(* PLC project SafeLOGIC-1, BrAutomation SafeDESIGNER  4.2.2.18 *)
(* stored: companyURL http://www.br-automation.com, creationDateTime Wed Apr 19 11:53:29 2017 *)

PROGRAM Main
  VAR  (* added by the conversion: wires and edge detectors of the diagram *)
    _AND_S80_OUT : ANY;
  END_VAR

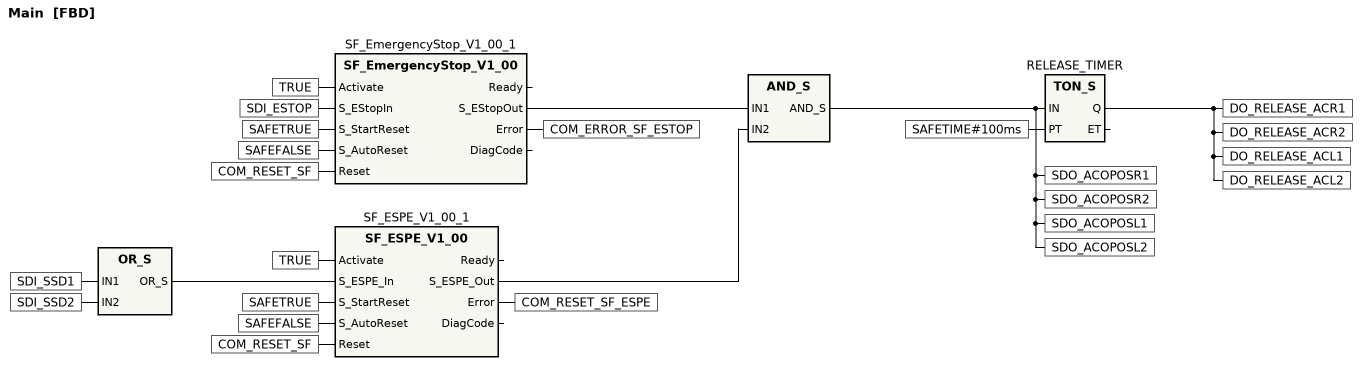
(* FBD diagram, written out as Structured Text *)
SF_EmergencyStop_V1_00_1(Activate := TRUE, S_EStopIn := SDI_ESTOP, S_StartReset := SAFETRUE, S_AutoReset := SAFEFALSE, Reset := COM_RESET_SF);
COM_ERROR_SF_ESTOP := SF_EmergencyStop_V1_00_1.Error;
SF_ESPE_V1_00_1(Activate := TRUE, S_ESPE_In := OR_S(SDI_SSD1, SDI_SSD2), S_StartReset := SAFETRUE, S_AutoReset := SAFEFALSE, Reset := COM_RESET_SF);
_AND_S80_OUT := AND_S(SF_EmergencyStop_V1_00_1.S_EStopOut, SF_ESPE_V1_00_1.S_ESPE_Out);
SDO_ACOPOSR1 := _AND_S80_OUT;
SDO_ACOPOSR2 := _AND_S80_OUT;
SDO_ACOPOSL1 := _AND_S80_OUT;
SDO_ACOPOSL2 := _AND_S80_OUT;
RELEASE_TIMER(IN := _AND_S80_OUT, PT := SAFETIME#100ms);
DO_RELEASE_ACR1 := RELEASE_TIMER.Q;
DO_RELEASE_ACR2 := RELEASE_TIMER.Q;
COM_RESET_SF_ESPE := SF_ESPE_V1_00_1.Error;
DO_RELEASE_ACL1 := RELEASE_TIMER.Q;
DO_RELEASE_ACL2 := RELEASE_TIMER.Q;
END_PROGRAM
